    # this is the main entry point for calculations, for Cover Corner.
    # it takes in the 4 touchpoints, analyzes the shape of the box.
    # returns the pathpoints
    # specifically for Around and Down then Straight (AtS)
    # specifically for left-sided boxes (vertical weld on left side of edge)
    def main_calculate_cover(p11, p12, p21, p3, leftwallthick, rightwallthick, leftchoice):
        struct1 = analyze_touchpoints_only_cover(p11, p12, p21, p3)
        if leftchoice:
            struct2 = calculate_AtS_points_cover_left(struct1, leftwallthick, rightwallthick)
        else:
            struct2 = calculate_AtS_points_cover_right(struct1, leftwallthick, rightwallthick)
        end
        #struct2 = calculate_DOtA_points_left_extended(struct1, list1, chamferover, chamferup, tcp_pose_top)
        #struct3 = check_validity_left(struct1, struct2)
        return struct2
    end

    def calculate_AtS_points_cover_left(struct1, leftwallthick, rightwallthick):
        # get the stuff from the struct
        pointintersect = struct1[0]
        heading1 = struct1[1]
        heading2 = struct1[2]
        heading3 = struct1[3]
        l1delxunit = struct1[4]
        l1delyunit = struct1[5]
        l2delxunit = struct1[6]
        l2delyunit = struct1[7]

        # FIND THE POINTS ON THE LINES OF THE FIRST TURN PATH
        # find locations 8 inches away from  intersect point
        # CONST
        welddistance1 = 6 # first path first leg (down)
        welddistance2 = 4 # first path second leg (under) # inches
        welddistance3 = 6 # second path (back away) # inches

        wd1 = welddistance1 * 25.4 / 1000
        wd2 = welddistance2 * 25.4 / 1000
        wd3 = welddistance3 * 25.4 / 1000
        leftwallthickmm = leftwallthick * 25.4 / 1000 # in this step corner right, this is distance from left edge
        rightwallthickmm =  rightwallthick * 25.4 / 1000 # in this step corner right, this is distance from right edge

        # first, check if we need a lift column raise
        # (we do, because for maximum reach we want to make the lift pedestal be even with the top of the covers)
        zpi = pointintersect[2]
        if zpi > 0:
            liftcolumnzneeded = zpi * 1000.0 # the robot uses coordinates in meters, but the lift column uses coordinates in mm
            z = 0
        else:
            z = zpi
        end

        # first, calculate the location of the top of the vertical chamfer (where point2 would be if there weren't any circle motion)
        x = pointintersect[0] + l2delxunit * rightwallthickmm
        y = pointintersect[1] + l2delyunit * rightwallthickmm
        #z = pointintersect[2] # replaced by z of lift column (directly above)
        pointtopvcham = p[x, y, z, 0, 0, 0]

        # calculate the rxryrz for the gun when it's at point1
        # start with rxryrz = 0,0,0 (gun facing up, preheat facing y+ axis.
        # rotate it 180 degrees about x axis. gun facing down, preheat facing y- axis
        # rotate it about 45 degrees ccw about z axis. x+ to heading1 is about 135 degrees. so our angle is heading1 - 90 degrees
        m1 = get_rotation_matrix_from_description("x", -1, 180 * pi / 180) # rotation 1: 180 degrees forward about x axis
        m2 = get_rotation_matrix_from_description("z", 1, heading1 - pi/2) # rotation 2
        m3 = multiply_matrix(m2, m1) #we rotate m1 first then m2, so we multiply in backwards order: 2 then 1
        rxryrz = convert_matrix_to_axang(m3)
        rx = rxryrz[0]
        ry = rxryrz[1]
        rz = rxryrz[2]

        # next, calculate point1
        p1x = x + l1delxunit * wd1
        p1y = y + l1delyunit * wd1
        point1 = p[p1x, p1y, z, rx, ry, rz]

        # the round over distance is the distance from pointbottomvcham to point2 (which will be the same as distance to p4)
        roundoverdistance = 0.05
        rod = roundoverdistance * 25.4 / 1000
        p2x = x + l1delxunit * rod
        p2y = y + l1delyunit * rod
        point2 = p[p2x, p2y, z, rx, ry, rz]

        # calculate the rxryrz for facing the down the left side of the box
        # rotate about x 90 (forward). then rotate about z ~ 45 (ccw)
        m1 = get_rotation_matrix_from_description("x", -1, 90 * pi / 180)
        m2 = get_rotation_matrix_from_description("z", 1, heading1 - pi/2)
        m3 = multiply_matrix(m2, m1) #we rotate m1 first then m2, so we multiply in backwards order: 2 then 1
        rxryrz = convert_matrix_to_axang(m3)
        rx = rxryrz[0]
        ry = rxryrz[1]
        rz = rxryrz[2]

        # calculate point4
        point4 = p[x, y, z - rod, rx, ry, rz]

        # calculate point5
        point5 = p[x, y, z - wd2, rx, ry, rz]

        # calculate point3
        # we know that the angle is exactly 90 degrees
        delta = calc_rod_midpoint_90deg(rod)
        p3z = z - delta
        p3x = x + delta * l1delxunit
        p3y = y + delta * l1delyunit

        # calculate rxryrz
        m1 = get_rotation_matrix_from_description("x", -1, 135 * pi / 180) # rotation 1: 135 degrees forward about x axis
        m2 = get_rotation_matrix_from_description("z", 1, heading1 - pi/2)
        m3 = multiply_matrix(m2, m1) #we rotate m1 first then m2, so we multiply in backwards order: 2 then 1
        rxryrz = convert_matrix_to_axang(m3)
        rx = rxryrz[0]
        ry = rxryrz[1]
        rz = rxryrz[2]
        point3 = p[p3x, p3y, p3z, rx, ry, rz]

        #todo: calculate trail out point

        # calculate back-away (points 201 and 202)
        pushtipforward = 0.006 # 6 millimeters forward. the tip needs to clear the capping wall's angled chamfer to not BONK when getting into position
        p201x = x + l1delxunit * leftwallthickmm + l2delxunit * pushtipforward
        p201y = y + l1delyunit * leftwallthickmm + l2delyunit * pushtipforward

        # calculate rxryrz
        # rotate 180 degrees about x. then rotate (90 deg + heading3 degrees) about z ccw
        m1 = get_rotation_matrix_from_description("x", -1, 180 * pi / 180)
        m2 = get_rotation_matrix_from_description("z", 1, heading3 + pi/2)
        m3 = multiply_matrix(m2, m1) #we rotate m1 first then m2, so we multiply in backwards order: 2 then 1
        rxryrz = convert_matrix_to_axang(m3)
        rx = rxryrz[0]
        ry = rxryrz[1]
        rz = rxryrz[2]
        point201 = p[p201x, p201y, z, rx, ry, rz]

        # calculate point 201's preheat
        pushtipforward2 = 0.012 - pushtipforward # 12 mm forward to clear the existing extrudant (but still have the extrudant from this extrusion join the existing). subtract from previous to make it constant even if you change pushtipforward1
        preheatdistance = 0.010 # 10 mm . above what it would be pushed down
        point201a = p[p201x, p201y, z + preheatdistance, rx, ry, rz]
        p201bx = p201x + l2delxunit * pushtipforward2
        p201by = p201y + l2delyunit * pushtipforward2
        point201b = p[p201bx, p201by, z + preheatdistance, rx, ry, rz]
        point201c = p[p201bx, p201by, z, rx, ry, rz]

        # calculate point 202
        p202x = p201x + wd3 * l2delxunit
        p202y = p201y + wd3 * l2delyunit
        point202 = p[p202x, p202y, z, rx, ry, rz]

        struct2 = struct(point1=point1, point2=point2, point3=point3, point4=point4, point5=point5, point201=point201, point202=point202, point201a=point201a, point201b=point201b, point201c=point201c)
        return struct2
    end

    def calculate_AtS_points_cover_right(struct1, leftwallthick, rightwallthick):
        # get the stuff from the struct
        pointintersect = struct1[0]
        heading1 = struct1[1]
        heading2 = struct1[2]
        heading3 = struct1[3]
        l1delxunit = struct1[4]
        l1delyunit = struct1[5]
        l2delxunit = struct1[6]
        l2delyunit = struct1[7]

        # FIND THE POINTS ON THE LINES OF THE FIRST TURN PATH
        # find locations 8 inches away from  intersect point
        # CONST
        welddistance1 = 6 # first path first leg (down)
        welddistance2 = 4 # first path second leg (under) # inches
        welddistance3 = 6 # second path (back away) # inches

        wd1 = welddistance1 * 25.4 / 1000
        wd2 = welddistance2 * 25.4 / 1000
        wd3 = welddistance3 * 25.4 / 1000
        leftwallthickmm = leftwallthick * 25.4 / 1000 # in this step corner right, this is distance from left edge
        rightwallthickmm =  rightwallthick * 25.4 / 1000 # in this step corner right, this is distance from right edge

        # first, check if we need a lift column raise
        # (we do, because for maximum reach we want to make the lift pedestal be even with the top of the covers)
        zpi = pointintersect[2]
        if zpi > 0:
            liftcolumnzneeded = zpi * 1000.0 # the robot uses coordinates in meters, but the lift column uses coordinates in mm
            z = 0
        else:
            z = zpi
        end

        # first, calculate the location of the top of the vertical chamfer (where point2 would be if there weren't any circle motion)
        x = pointintersect[0] + l1delxunit * leftwallthickmm
        y = pointintersect[1] + l1delyunit * leftwallthickmm
        #z = pointintersect[2] # replaced by z of lift column (directly above)
        pointtopvcham = p[x, y, z, 0, 0, 0]

        # calculate the rxryrz for the gun when it's at point1
        # start with rxryrz = 0,0,0 (gun facing up, preheat facing y+ axis.
        # rotate it 180 degrees about x axis. gun facing down, preheat facing y- axis
        # rotate it about 135 degrees ccw about z axis. x+ to heading3 is about 225 degrees. so our angle is heading3 - 90 degrees
        m1 = get_rotation_matrix_from_description("x", -1, 180 * pi / 180) # rotation 1: 180 degrees forward about x axis
        m2 = get_rotation_matrix_from_description("z", 1, heading3 - pi/2) # rotation 2
        m3 = multiply_matrix(m2, m1) #we rotate m1 first then m2, so we multiply in backwards order: 2 then 1
        rxryrz = convert_matrix_to_axang(m3)
        rx = rxryrz[0]
        ry = rxryrz[1]
        rz = rxryrz[2]

        # next, calculate point1
        p1x = x + l2delxunit * wd1
        p1y = y + l2delyunit * wd1
        point1 = p[p1x, p1y, z, rx, ry, rz]

        # the round over distance is the distance from pointbottomvcham to point2 (which will be the same as distance to p4)
        roundoverdistance = 0.05
        rod = roundoverdistance * 25.4 / 1000
        p2x = x + l2delxunit * rod
        p2y = y + l2delyunit * rod
        point2 = p[p2x, p2y, z, rx, ry, rz]

        # calculate the rxryrz for facing the down the right side of the box
        # rotate about x 90 (forward). then rotate about z ~ 135 (ccw)
        m1 = get_rotation_matrix_from_description("x", -1, 90 * pi / 180)
        m2 = get_rotation_matrix_from_description("z", 1, heading3 - pi/2)
        m3 = multiply_matrix(m2, m1) #we rotate m1 first then m2, so we multiply in backwards order: 2 then 1
        rxryrz = convert_matrix_to_axang(m3)
        rx = rxryrz[0]
        ry = rxryrz[1]
        rz = rxryrz[2]

        # calculate point4
        point4 = p[x, y, z - rod, rx, ry, rz]

        # calculate point5
        point5 = p[x, y, z - wd2, rx, ry, rz]

        # calculate point3
        # we know that the angle is exactly 90 degrees
        delta = calc_rod_midpoint_90deg(rod)
        p3z = z - delta
        p3x = x + delta * l2delxunit
        p3y = y + delta * l2delyunit

        # calculate rxryrz
        m1 = get_rotation_matrix_from_description("x", -1, 135 * pi / 180) # rotation 1: 135 degrees forward about x axis
        m2 = get_rotation_matrix_from_description("z", 1, heading3 - pi/2)
        m3 = multiply_matrix(m2, m1) #we rotate m1 first then m2, so we multiply in backwards order: 2 then 1
        rxryrz = convert_matrix_to_axang(m3)
        rx = rxryrz[0]
        ry = rxryrz[1]
        rz = rxryrz[2]
        point3 = p[p3x, p3y, p3z, rx, ry, rz]

        #todo: calculate trail out point

        # calculate back-away (points 201 and 202)
        pushtipforward = 0.006 # 6 millimeters forward. the tip needs to clear the capping wall's angled chamfer to not BONK when getting into position
        p201x = x + l2delxunit * rightwallthickmm + l1delxunit * pushtipforward
        p201y = y + l2delyunit * rightwallthickmm + l1delyunit * pushtipforward

        # calculate rxryrz
        # rotate 180 degrees about x. then rotate (90 deg + heading1 degrees) about z ccw
        m1 = get_rotation_matrix_from_description("x", -1, 180 * pi / 180)
        m2 = get_rotation_matrix_from_description("z", 1, heading1 + pi/2)
        m3 = multiply_matrix(m2, m1) #we rotate m1 first then m2, so we multiply in backwards order: 2 then 1
        rxryrz = convert_matrix_to_axang(m3)
        rx = rxryrz[0]
        ry = rxryrz[1]
        rz = rxryrz[2]
        point201 = p[p201x, p201y, z, rx, ry, rz]

        # calculate point 201's preheat
        pushtipforward2 = 0.012 - pushtipforward # 12 mm forward to clear the existing extrudant (but still have the extrudant from this extrusion join the existing). subtract from previous to make it constant even if you change pushtipforward1
        preheatdistance = 0.010 # 10 mm . above what it would be pushed down
        point201a = p[p201x, p201y, z + preheatdistance, rx, ry, rz]
        p201bx = p201x + l1delxunit * pushtipforward2
        p201by = p201y + l1delyunit * pushtipforward2
        point201b = p[p201bx, p201by, z + preheatdistance, rx, ry, rz]
        point201c = p[p201bx, p201by, z, rx, ry, rz]

        # calculate point 202
        p202x = p201x + wd3 * l1delxunit
        p202y = p201y + wd3 * l1delyunit
        point202 = p[p202x, p202y, z, rx, ry, rz]

        struct2 = struct(point1=point1, point2=point2, point3=point3, point4=point4, point5=point5, point201=point201, point202=point202)
        return struct2
    end
    $ 9 "pathturn≔main_calculate_cover(p11,p12,p21,p3fh,.628,.375, True )"
    global pathturn=main_calculate_cover(p11,p12,p21,p3fh,.628,.375,  True  )
    $ 10 "Comment"
    # Comment
    $ 11 "align_for_cover_left()"
    align_for_cover_left()
    $ 12 "Set"
    set_tcp(p[0.00451,-0.328,0.10573,1.2092,-1.2092,1.2092])
    $ 13 "Comment"
    # Comment
    $ 14 "p1≔pathturn[0]"
    global p1=pathturn[0]
    $ 15 "p2≔pathturn[1]"
    global p2=pathturn[1]
    $ 16 "p3≔pathturn[2]"
    global p3=pathturn[2]
    $ 17 "p4≔pathturn[3]"
    global p4=pathturn[3]
    $ 18 "p5≔pathturn[4]"
    global p5=pathturn[4]
    $ 19 "pa1≔p[p1[0],p1[1],p1[2]+0.05,p1[3],p1[4],p1[5]]"
    global pa1=p[p1[0],p1[1],p1[2]+0.05,p1[3],p1[4],p1[5]]
    $ 20 "MoveJ"
    $ 21 "pa1" "breakAfter"
    movej(pa1, a=1.3962634015954636, v=1.0471975511965976)
    $ 22 "MoveL"
    $ 23 "p1" "breakAfter"
    movel(p1, a=0.05, v=0.05)
    $ 24 "Wait: 8.0"
    sleep(8.0)
    $ 25 "turn ext on"
    # begin: URCap Program Node
    #   Source: WireTank Serial, 4.9.0, WireTank, LLC
    #   Type: WireTank Serial
    $ 26 "Serial Bridge uR1"
    SerialResponse = WTSerialBridge.send_command("/dev/ttyUSB0",1200, 8, "None", "One", "None", 1000, "None", "None", [252,82,49], False)
    # end: URCap Program Node
    # begin: URCap Program Node
    #   Source: WireTank Serial, 4.9.0, WireTank, LLC
    #   Type: WireTank Serial
    $ 27 "Serial Bridge uR1"
    SerialResponse = WTSerialBridge.send_command("/dev/ttyUSB0",1200, 8, "None", "One", "None", 1000, "None", "None", [252,82,49], False)
    # end: URCap Program Node
    $ 28 "Wait: 1.0"
    sleep(1.0)
    $ 30 "Set DO[0]=On"
    set_standard_digital_out(0, True)
    $ 31 "MoveL"
    $ 32 "p2" "breakAfter"
    movel(p2, a=0.1, v=0.01)
    $ 34 "MoveP"
    $ 35 "CircleMove"
    $ 36 "p3" "noBreak"

    $ 37 "p4" "breakAfter"
    movec(p3, p4, a=0.01, v=5.0E-4, r=0.001, mode=1)
    $ 39 "MoveL"
    $ 40 "p5" "breakAfter"
    movel(p5, a=0.05, v=0.012)
    # begin: URCap Program Node
    #   Source: WireTank Serial, 4.9.0, WireTank, LLC
    #   Type: WireTank Serial
    $ 41 "Serial Bridge uR0"
    SerialResponse = WTSerialBridge.send_command("/dev/ttyUSB0",1200, 8, "None", "One", "None", 1000, "None", "None", [252,82,48], False)
    # end: URCap Program Node
    $ 42 "Wait: 2.0"
    sleep(2.0)
    $ 43 "Set DO[0]=Off"
    set_standard_digital_out(0, False)
    $ 44 "Comment"
    # Comment
    $ 45 "pret1≔p[p5[0]+0.05,p5[1],p5[2],p5[3],p5[4],p5[5]]"
    global pret1=p[p5[0]+0.05,p5[1],p5[2],p5[3],p5[4],p5[5]]
    $ 46 "pret2≔p[p5[0]+0.1,p5[1],p5[2]+0.2,p5[3],p5[4],p5[5]]"
    global pret2=p[p5[0]+0.1,p5[1],p5[2]+0.2,p5[3],p5[4],p5[5]]
    $ 53 "p201≔pathturn[5]"
    global p201=pathturn[5]
    $ 54 "p202≔pathturn[6]"
    global p202=pathturn[6]
    $ 55 "p201a≔pathturn[7]"
    global p201a=pathturn[7]
    $ 56 "p201b≔pathturn[8]"
    global p201b=pathturn[8]
    $ 57 "p201c≔pathturn[9]"
    global p201c=pathturn[9]
    $ 58 "pret3≔p[p201[0],p201[1],p201[2]+0.05,p201[3],p201[4],p201[5]]"
    global pret3=p[p201[0],p201[1],p201[2]+0.05,p201[3],p201[4],p201[5]]
    $ 59 "pret4≔p[p202[0],p202[1],p202[2]+0.05,p202[3],p202[4],p202[5]]"
    global pret4=p[p202[0],p202[1],p202[2]+0.05,p202[3],p202[4],p202[5]]
    $ 63 "Set"
    set_tcp(p[-0.0095,-0.328,0.10573,1.2092,-1.2092,1.2092])
    $ 64 "MoveL"
    $ 65 "pret1" "breakAfter"
    movel(pret1, a=0.05, v=0.05)
    $ 66 "MoveJ"
    $ 67 "pret2" "breakAfter"
    movej(pret2, a=1.3962634015954636, v=1.0471975511965976)
    $ 68 "MoveJ"
    $ 69 "'retreat of p5'"
    # 'retreat of p5'
    $ 70 "Waypoint_1" "breakAfter"
    movej(get_inverse_kin(Waypoint_1_p, qnear=Waypoint_1_q), a=1.3962634015954636, v=1.0471975511965976)
    $ 74 "MoveJ"
    $ 75 "'requires a shoulder flip. safe waypoints for that:'"
    # 'requires a shoulder flip. safe waypoints for that:'
    $ 76 "Waypoint_3" "breakAfter"
    movej(get_inverse_kin(Waypoint_3_p, qnear=Waypoint_3_q), a=1.3962634015954636, v=1.0471975511965976)
    $ 77 "Waypoint_4" "breakAfter"
    movej(get_inverse_kin(Waypoint_4_p, qnear=Waypoint_4_q), a=1.3962634015954636, v=1.0471975511965976)
    $ 78 "MoveJ"
    $ 79 "'approach of p201'"
    # 'approach of p201'
    $ 80 "Waypoint_2" "breakAfter"
    movej(get_inverse_kin(Waypoint_2_p, qnear=Waypoint_2_q), a=1.3962634015954636, v=1.0471975511965976)
    $ 81 "MoveJ"
    $ 82 "pret3" "breakAfter"
    movej(pret3, a=1.3962634015954636, v=1.0471975511965976)
    $ 83 "MoveL"
    $ 85 "p201a" "breakAfter"
    movel(p201a, a=0.05, v=0.05)
    $ 86 "Wait: 6.0"
    sleep(6.0)
    $ 87 "MoveL"
    $ 88 "p201b" "breakAfter"
    movel(p201b, a=1.2, v=0.01)
    $ 89 "p201c" "breakAfter"
    movel(p201c, a=1.2, v=0.01)
    $ 90 "turn ext on"
    # begin: URCap Program Node
    #   Source: WireTank Serial, 4.9.0, WireTank, LLC
    #   Type: WireTank Serial
    $ 91 "Serial Bridge uR1"
    SerialResponse = WTSerialBridge.send_command("/dev/ttyUSB0",1200, 8, "None", "One", "None", 1000, "None", "None", [252,82,49], False)
    # end: URCap Program Node
    # begin: URCap Program Node
    #   Source: WireTank Serial, 4.9.0, WireTank, LLC
    #   Type: WireTank Serial
    $ 92 "Serial Bridge uR1"
    SerialResponse = WTSerialBridge.send_command("/dev/ttyUSB0",1200, 8, "None", "One", "None", 1000, "None", "None", [252,82,49], False)
    # end: URCap Program Node
    $ 93 "Wait: 1.0"
    sleep(1.0)
    $ 95 "Set DO[0]=On"
    set_standard_digital_out(0, True)
    $ 96 "MoveL"
    $ 97 "p202" "breakAfter"
    movel(p202, a=0.1, v=0.012)
    # begin: URCap Program Node
    #   Source: WireTank Serial, 4.9.0, WireTank, LLC
    #   Type: WireTank Serial
    $ 98 "Serial Bridge uR0"
    SerialResponse = WTSerialBridge.send_command("/dev/ttyUSB0",1200, 8, "None", "One", "None", 1000, "None", "None", [252,82,48], False)
    # end: URCap Program Node
    $ 99 "Wait: 2.0"
    sleep(2.0)
    $ 100 "Set DO[0]=Off"
    set_standard_digital_out(0, False)
    $ 101 "MoveJ"
    $ 102 "pret4" "breakAfter"
    movej(pret4, a=1.3962634015954636, v=1.0471975511965976)
    $ 103 "MoveJ"
    $ 104 "Waypoint_2" "breakAfter"
    movej(get_inverse_kin(Waypoint_2_p, qnear=Waypoint_2_q), a=1.3962634015954636, v=1.0471975511965976)
    $ 105 "Home"
    movej([-3.266929759358355, -1.2139462677784536, 1.5878387874396154, 1.1069165929565088, -0.0023738326664366483, -1.7891447305770605], a=1.3962634015954636, v=1.0471975511965976)
    # begin: URCap Program Node
    #   Source: MachineLogic for Universal Robots, 3.1.7, Vention Inc.
    #   Type: MachineLogic for Universal Robots
    $ 106 "MachineLogic Homing"
    while isVentionMovementBusyMachineMotion1==True:
    sleep(0.05)
    end
    if(isVentionMovementBusyMachineMotion1 == False):
    isVentionMovementBusyMachineMotion1 = True
    socket_send_string("estop/status;", "MachineMotion1")
    temp_estop_var_vention = socket_read_string("MachineMotion1",timeout=15)
    while(temp_estop_var_vention=="estop/status true"):
    if temp_estop_var_vention=="estop/status true":
    sendStringWithTimeout("estop/systemreset/request","Ack estop/systemreset/request;","MachineMotion1")
    end
    socket_send_string("estop/status;", "MachineMotion1")
    temp_estop_var_vention = socket_read_string("MachineMotion1",timeout=15)
    if temp_estop_var_vention=="estop/status true":
    popup("MachineMotion in estop, make sure you have all emergency modules released manually. If you continue the system will try to reset MachineMotion automatically.",blocking=True)
    end
    end
    else:
    popup("resource is being used already: MachineMotion1")
    halt
    end
    isVentionMovementBusyMachineMotion1 = True
    sendString("im_home_axis_1", "MachineMotion im_home_axis_1 = completed", "MachineMotion1")
    isVentionMovementBusyMachineMotion1 = False
    sendString("SET im_set_encoder_pos_aux_1 0.000", "Ack", "MachineMotion1")
    isVentionMovementBusyMachineMotion1 = False
    sleep(0.03)
    # end: URCap Program Node
  end
end
